Fanuc KAREL source: MP0085.KL

PROGRAM MP0085
%STACKSIZE=65535
%PRIORITY=65535
%NOLOCKGROUP
ROUTINE FINT(P1 : INTEGER) : INTEGER FROM MP0085
ROUTINE FREAL(P1 : REAL) : REAL FROM MP0085
ROUTINE RTEST(P1 : INTEGER; P2 : REAL) FROM MP0085
ROUTINE FINT
BEGIN
RETURN((P1 + 1))
END FINT
ROUTINE FREAL
BEGIN
RETURN((P1 + 1.0))
END FREAL
ROUTINE RTEST
VAR
S1 : INTEGER
U2C_2 : INTEGER
U2C_3 : INTEGER
U2C_4 : REAL
U2C_5 : REAL
U2C_6 : REAL
U2C_7 : INTEGER
U2C_8 : REAL
BEGIN
S1=7
U2C_2=3
U2C_3=2
U2C_4=2.5
U2C_5=4.5
U2C_6=1.5
-- UNSAFE_SOURCE_IR line 28: CALL_RESULT FINT(S1)
END RTEST
BEGIN
RTEST(7,2.5)
END MP0085
